(* CoDeSys 2.3 export: HOL_PARTER.EXP *)

(* POU Rooms/Hol_parter, ST *)
FUNCTION_BLOCK Hol_parter
VAR
	lampNextToL:OnOff;
(*	lampNextToE:OnOff; *)
	mainLamp:OnOff;

	tmp: BOOL;
END_VAR
mainLamp(input:=H9_2a, output => H7_1);

lampNextToL(input:=H9_2b OR H3_1a);
H1_1:= lampNextToL.state;
H6_1:=lampNextToL.state;
END_FUNCTION_BLOCK
